ABB RobotStudio station: LoadingAreaV2_1.rsstn

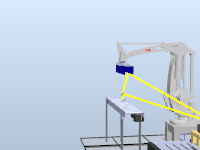
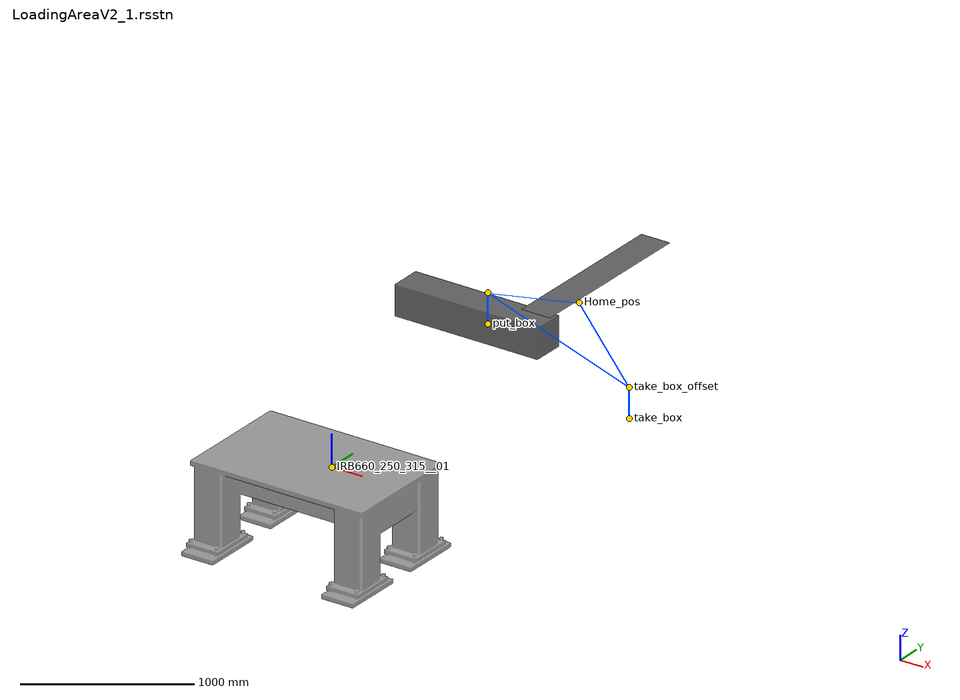
[picture v1: parts stored in the station drawn from their meshes, with robot base, taught points and paths (robot models come from the ABB library and are not in the file)]
Station LoadingAreaV2 (saved by RobotStudio 21.2.9526.0)
Controller IRB660_250_315
  mechanical unit ROB_1: IRB660_250_315__01, 6 joints, base frame (0, 0, 570) mm
Layout (positions relative to the parent item):
  - IRB660_250_315__01 [mechanism, from Robots\IRB660_250_315__01.rslib] at (0, 0, 570) mm; joint values [0, 0, 0, 0] (rad or m)
  - conv_box_top [part, from библиотеки\conv_box_top.rslib] at (1800, -500, 1316.27) mm
  - conv_pallets_top [part, from вариант 2\conv_pallets_top.rslib] at (-2942.14, 1371.97, 435) mm, rotated rx 0 ry 0 rz 90 deg
  - pallet [part, from вариант 2\pallet.rslib] at (427.78, 2270.2, 414.36) mm, rotated rx 0 ry -90 rz 90 deg
  - IRC5_Control-Module [part, from Equipment\IRC5_Control-Module.rslib] at (-1099.11, 0, 100) mm, rotated rx 90 ry 0 rz 90 deg
  - Стол [part] at (445, -335, 540) mm, rotated rx 90 ry 0 rz 90 deg, size 980 x 570 x 1200 mm
  - Block [part] at (-382.22, 3740.2, -624.64) mm, rotated rx 0 ry 0 rz -90 deg, size 210 x 1000 x 200 mm
  - Gripper [mechanism] at (1910, 0, 2403) mm, rotated rx 180 ry 0 rz 180 deg; joint values [-0.0498] (rad or m)
      TCP Gripper_1 at (178, 0, 299) mm
      links: L1, L2
  - Attacher [part] at (1950, -605, 2310) mm, rotated rx 0 ry 90 rz 0 deg, size 0 x 1200 x 200 mm
Attachment: Gripper is attached to IRB660_250_315__01 / Link6
Attachment: Attacher is attached to IRB660_250_315__01 / Link6
EventTableEntry 1033: Group=, Trigger=doOpenGripper 1034, Actions=[EventTableActionMechanicalPose 1035], Comment=, ActivationMode=2, Cyclic=false
EventTableTriggerIO 1034: IOValue=[1], IRC5Controller=? -1, Operator=0, SignalSource=IRB660_250_315 515
EventTableActionMechanicalPose 1035: VirtualSignal=, Mechanism=Gripper 1028, ToPoseName=HomePosition, VirtualSignalValue=[1]
EventTableEntry 1036: Group=, Trigger=doCloseGripper 1037, Actions=[EventTableActionMechanicalPose 1038], Comment=, ActivationMode=2, Cyclic=false
EventTableTriggerIO 1037: IOValue=[1], IRC5Controller=? -1, Operator=0, SignalSource=IRB660_250_315 515
EventTableActionMechanicalPose 1038: VirtualSignal=, Mechanism=Gripper 1028, ToPoseName=Pose_Closed, VirtualSignalValue=[1]
EventTableEntry 1039: Group=, Trigger=Attach 1040, Actions=[EventTableActionAttach 1041], Comment=, ActivationMode=2, Cyclic=false
EventTableTriggerIO 1040: IOValue=[1], IRC5Controller=? -1, Operator=0, SignalSource=IRB660_250_315 515
EventTableActionAttach 1041: AttachmentParent=Attacher 1183, AttachmentChild=Block 1023, MountObject=false, Offset=[X=1, Y=0, Z=0, W=0, X=0, Y=1, Z=0, W=0, X=0, Y=0, Z=1, W=0, X=0, Y=0, Z=0, W=1], FlangeIndext=0, FindNearest=false
EventTableEntry 1042: Group=, Trigger=Detach 1043, Actions=[EventTableActionDetach 1044], Comment=, ActivationMode=2, Cyclic=false
EventTableTriggerIO 1043: IOValue=[1], IRC5Controller=? -1, Operator=0, SignalSource=IRB660_250_315 515
EventTableActionDetach 1044: AttachmentParent=Attacher 1183, AttachmentChild=Block 1023
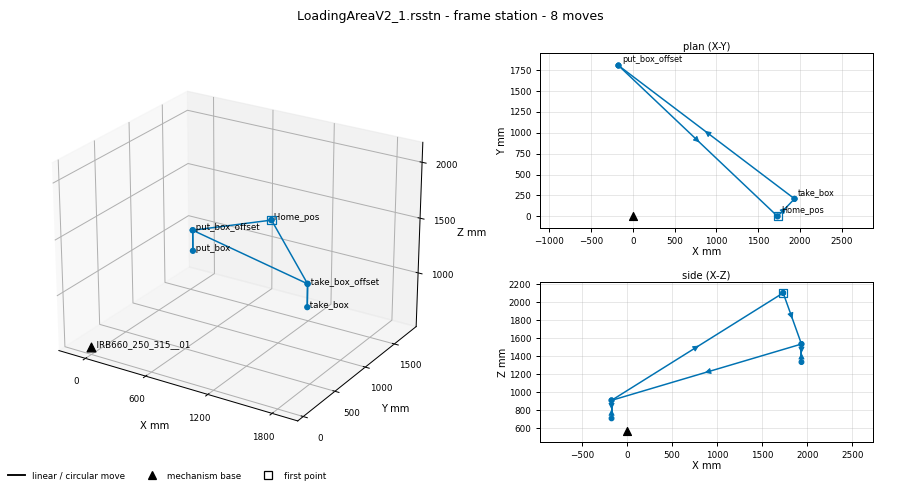
[picture p0: tool path of LoadingAreaV2_1.rsstn in frame station, 8 of 8 moves have a stored position in this frame; points joined in program order, loops and branches not executed]
Targets, tools, work objects and paths stored in the station, written as RAPID:
! task T_ROB1
MODULE CalibData
  PERS tooldata Gripper_1:=[TRUE,[[178,0,299],[1,0,0,0]],[2.5,[0,0,100],[1,0,0,0],0,0,0]];
  TASK PERS wobjdata Wobj_box:=[FALSE,TRUE,"",[[0,0,0],[1,0,0,0]],[[0,0,0],[1,0,0,0]]];
  TASK PERS wobjdata Wobj_pallet:=[FALSE,TRUE,"",[[427.78,1470.197,414.355],[0.707106781,0,0,0.707106781]],[[0,0,0],[1,0,0,0]]];
ENDMODULE

! task T_ROB1
MODULE Module1
  CONST robtarget take_box:=[[1935,210,1337],[0,0,1,0],[0,0,0,0],[9E+09,9E+09,9E+09,9E+09,9E+09,9E+09]];
  CONST robtarget put_box:=[[335,600,298],[0,1,0,0],[0,0,0,0],[9E+09,9E+09,9E+09,9E+09,9E+09,9E+09]];
  CONST robtarget take_box_offset:=[[1935,210,1537],[0,0,1,0],[0,0,0,0],[9E+09,9E+09,9E+09,9E+09,9E+09,9E+09]];
  CONST robtarget put_box_offset:=[[335,600,498],[0,1,0,0],[0,0,0,0],[9E+09,9E+09,9E+09,9E+09,9E+09,9E+09]];
  CONST robtarget Home_pos:=[[1732,0,2104],[0,0,1,0],[0,0,0,0],[9E+09,9E+09,9E+09,9E+09,9E+09,9E+09]];
  PROC Path_10()
    MoveL Home_pos,v1000,z100,Gripper_1\WObj:=wobj0;
    MoveL take_box_offset,v1000,z100,Gripper_1\WObj:=Wobj_box;
    MoveL take_box,v1000,z100,Gripper_1\WObj:=Wobj_box;
    MoveL take_box_offset,v1000,z100,Gripper_1\WObj:=Wobj_box;
    MoveL put_box_offset,v1000,z100,Gripper_1\WObj:=Wobj_pallet;
    MoveL put_box,v1000,z100,Gripper_1\WObj:=Wobj_pallet;
    MoveL put_box_offset,v1000,z100,Gripper_1\WObj:=Wobj_pallet;
    MoveL Home_pos,v1000,z100,Gripper_1\WObj:=wobj0;
  ENDPROC
ENDMODULE

